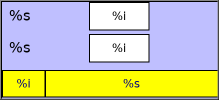
VISUALIZATION VISU_CR_SW_GENIUS_ETH  // 219x100
VAR_IN_OUT
	m_Input_BALAYAGE : BLOCK_IND_CREUSET_GENIUS_ETHERCAT;
END_VAR
    Rectangle (0,0 219x100)
    Rectangle (6,1 118x29), "%s", text list: 'TextList_Evap', text index: 0
    Rectangle (2,70 43x27), "%i", text variable: m_Input_BALAYAGE.STATE_POS_CR
    Rectangle (45,70 173x27), "%s", text variable: m_Input_BALAYAGE.STATE_MAT
    RoundedRectangle (89,2 60x28), "%i", text variable: m_Input_BALAYAGE.PRM_NCR, input disabled if: NOT Global_Variables.PRG_USER.ACTU_USER.MAINTENANCE OR NOT MACHINE.STATE_Manu
        OnMouseDown: write the text variable via VisuDialogs.Numpad, min 1, max m_Input_BALAYAGE.CONF_NCR
    Rectangle (6,33 118x29), "%s", text list: 'TextList_Evap', text index: 1
    RoundedRectangle (89,34 60x28), "%i", text variable: m_Input_BALAYAGE.PRM_NBAL, input disabled if: NOT Global_Variables.PRG_USER.ACTU_USER.MAINTENANCE OR NOT MACHINE.STATE_Manu
        OnMouseDown: write the text variable via VisuDialogs.Numpad, min 1, max 8
END_VISUALIZATION

(* stored: Version 1.1.0.1, ProductVersion 3.1.4024.10
   Visu VISU_CR_SW_GENIUS_ETH: Id {3f7b05a4-2544-462d-99e4-79e9186bdf6b} *)
